# EPICS substitutions: modules/event/evrSupport/Db/ioc/IOC-LI21-MG01evr.substitutions
#==============================================================================
#
# Abs:  LCLS EVR IOC records for LI21 MG01
#
# Name: IOC-LI21-MG01evr.substitutions
#
#==============================================================================
#
file evrMGXX.db
{
pattern { DEVICE        }
	{ EVR:LI21:MG01 }
}
